// TIA Portal V16 export
// export: Created 2022-06-11T10:19:43.8619966Z, ExportSetting WithDefaults, DisplayName Totally Integrated Automation Portal, DisplayVersion V16 Update 3, DisplayName TIA Portal Version Control Interface, DisplayVersion V16 Update 2, DisplayName TIA Portal Openness, DisplayVersion V16 Update 3, DisplayName STEP 7 Professional, DisplayVersion V16 Update 3, DisplayName STEP 7 Safety, DisplayVersion V16, DisplayName WinCC Professional, DisplayVersion V16 Update 3
TYPE "UT11011_St_DevValve3Way"
TITLE = Static UDT [DEVICE DRIVER] — Three-way Valve
// PRACTICAL SERIES AUTOMATION LIBRARY (PAL)   —   COPYRIGHT 2020 – M. GLEDHILL (MIT LICENCE)
//                   ———— ◆ ————
// FULL ONLINE DOCUMENTATION IS AVAILABLE AT: https://practicalseries.com/2001-pal/index.html
// stored: IsFailsafeCompliant false
   STRUCT
      revInfo { ExternalWritable := 'False'} : "UT01000_St_SysRevision";   // Revision information
      ___________0010_0 { ExternalAccessible := 'False'; ExternalVisible := 'False'; ExternalWritable := 'False'} : Int;
      ___________0010_1 { ExternalAccessible := 'False'; ExternalVisible := 'False'; ExternalWritable := 'False'} : Int;   // ▀▀▀▀ INSTRUMENT CONFIGURATION
      CONFIG_FBK_ENG_EN : Bool;   // CONFIG — Energised feedback is enabled (1 = ENG feedback present, 0 = no ENG feedback)
      CONFIG_FBK_DENG_EN : Bool;   // CONFIG — Deenergised feedback is enabled (1 = DENG feedback present, 0 = no DENG feedback)
      CONFIG_ESTOP_DIS : Bool;   // CONFIG — E_STOP signal disabled (1 = E_STOP not used, 0 = E_STOP in use)
      CONFIG_TRIP_DIS : Bool;   // CONFIG — TRIP signal disabled (1 = TRIP not used, 0 = TRIP in use)
      CONFIG_ILOCK_DIS : Bool;   // CONFIG — INTERLOCK signal disabled (1 = INTERLOCK not used, 0 = INTERLOCK in use)
      CONFIG_PERM_DIS : Bool;   // CONFIG — PERMISSIVE signal disabled (1 = PERMISSIVE not used, 0 = PERMISSIVE in use)
      CONFIG_TRIP_ENG_DENG : Bool;   // CONFIG — TRIP state (1 = energised if tripped, 0 = deenergised if tripped)
      CONFIG_ILOCK_ENG_DENG : Bool;   // CONFIG — INTERLOCK state (1 = energised if interlocked, 0 = deenergised if interlocked)
      CONFIG_PERM_ENG_DENG : Bool;   // CONFIG — PERMISSIVE permitted state (1 = permitted energised, 0 = permitted deenergised)
      CONFIG_FP_DIS { ExternalWritable := 'False'; S7_SetPoint := 'True'} : Bool;   // CONFIG — Faceplate is disabled (1 = no Faceplate, 0 = normal)
      CONFIG_MAN_DIS : Bool;   // CONFIG — Manual mode is disabled (1 = no manual mode – auto only, 0 = normal)
      CONFIG_BYPASS_DIS : Bool;   // CONFIG — Bypass mode is disabled (1 = no Bypass, 0 = normal)
      CONFIG_SIM_DIS { ExternalWritable := 'False'; S7_SetPoint := 'True'} : Bool;   // CONFIG — Simulation mode is disabled (1 = no Simulation, 0 = normal)
      CONFIG_RL_EN { ExternalWritable := 'False'; S7_SetPoint := 'True'} : Bool;   // CONFIG — Remote/local mode enabled (1 = remote/local permitted, 0 = remote/local N/A)
      ___________0020_0 { ExternalAccessible := 'False'; ExternalVisible := 'False'; ExternalWritable := 'False'} : Int;
      ___________0020_1 { ExternalAccessible := 'False'; ExternalVisible := 'False'; ExternalWritable := 'False'} : Int;   // ▀▀▀▀ INSTRUMENT INFORMATION (TAG & UNITS)
      INFO_TAG { ExternalWritable := 'False'; S7_SetPoint := 'True'} : String[20];   // INFORMATION — Instrument ID tag
      ___________0030_0 { ExternalAccessible := 'False'; ExternalVisible := 'False'; ExternalWritable := 'False'} : Int;
      ___________0030_1 { ExternalAccessible := 'False'; ExternalVisible := 'False'; ExternalWritable := 'False'} : Int;   // ▀▀▀▀ INSTRUMENT TIMER DEFAULT VALUES
      TIME_ENG_MAX { ExternalWritable := 'False'; S7_SetPoint := 'True'} : Real := 5.0;   // TIMER — Initial value of energising operation timer [seconds], counts down from this value
      TIME_DENG_MAX { ExternalWritable := 'False'; S7_SetPoint := 'True'} : Real := 5.0;   // TIMER — Initial value of deenergising operation timer [seconds], counts down from this value
      TIME_DER_ENG { ExternalWritable := 'False'; S7_SetPoint := 'True'} : Real := 95.0;   // TIMER — Percentage of energising timer to expired before derived ENG feedback [percentage]
      TIME_DER_DENG { ExternalWritable := 'False'; S7_SetPoint := 'True'} : Real := 95.0;   // TIMER — Percentage of deenergising timer to expired before derived DENG feedback [percentage]
   END_STRUCT;
   // revInfo.REV_BLOCK := 'UT11011';
   // revInfo.REV_NUMBER := '000.801';
   // revInfo.REV_DATE := '2022.06.07';
   // revInfo.REV_AUTHOR := 'M. Gledhill';
END_TYPE
